RESOURCE_TYPE FlexPRET
  (* Standard: 61499-2 *)
  (* Version 0.1, 2016-00-28, hpea485, UOA *)
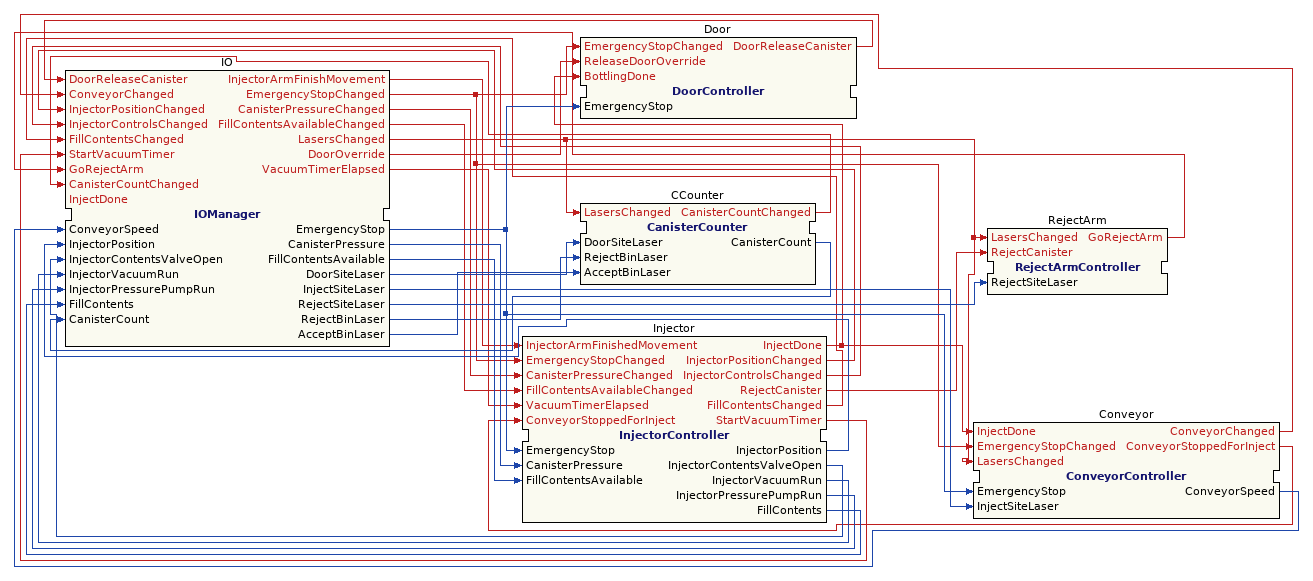
  FBS
    IO : IOManager;
    CCounter : CanisterCounter;
    Door : DoorController;
    Injector : InjectorController;
    Conveyor : ConveyorController;
    RejectArm : RejectArmController;
  END_FBS
  EVENT_CONNECTIONS
    IO.InjectorArmFinishMovement TO Injector.InjectorArmFinishedMovement;
    IO.EmergencyStopChanged TO Door.EmergencyStopChanged;
    IO.EmergencyStopChanged TO Injector.EmergencyStopChanged;
    IO.EmergencyStopChanged TO Conveyor.EmergencyStopChanged;
    IO.CanisterPressureChanged TO Injector.CanisterPressureChanged;
    IO.FillContentsAvailableChanged TO Injector.FillContentsAvailableChanged;
    IO.LasersChanged TO CCounter.LasersChanged;
    IO.LasersChanged TO RejectArm.LasersChanged;
    IO.LasersChanged TO Conveyor.LasersChanged;
    IO.DoorOverride TO Door.ReleaseDoorOverride;
    IO.VacuumTimerElapsed TO Injector.VacuumTimerElapsed;
    CCounter.CanisterCountChanged TO IO.CanisterCountChanged;
    Door.DoorReleaseCanister TO IO.DoorReleaseCanister;
    Injector.InjectDone TO Door.BottlingDone;
    Injector.InjectDone TO Conveyor.InjectDone;
    Injector.InjectorPositionChanged TO IO.InjectorPositionChanged;
    Injector.InjectorControlsChanged TO IO.InjectorControlsChanged;
    Injector.RejectCanister TO RejectArm.RejectCanister;
    Injector.FillContentsChanged TO IO.FillContentsChanged;
    Injector.StartVacuumTimer TO IO.StartVacuumTimer;
    Conveyor.ConveyorChanged TO IO.ConveyorChanged;
    Conveyor.ConveyorStoppedForInject TO Injector.ConveyorStoppedForInject;
    RejectArm.GoRejectArm TO IO.GoRejectArm;
  END_CONNECTIONS
  DATA_CONNECTIONS
    IO.EmergencyStop TO Door.EmergencyStop;
    IO.EmergencyStop TO Injector.EmergencyStop;
    IO.EmergencyStop TO Conveyor.EmergencyStop;
    IO.CanisterPressure TO Injector.CanisterPressure;
    IO.FillContentsAvailable TO Injector.FillContentsAvailable;
    IO.DoorSiteLaser TO CCounter.DoorSiteLaser;
    IO.InjectSiteLaser TO Conveyor.InjectSiteLaser;
    IO.RejectSiteLaser TO RejectArm.RejectSiteLaser;
    IO.RejectBinLaser TO CCounter.RejectBinLaser;
    IO.AcceptBinLaser TO CCounter.AcceptBinLaser;
    CCounter.CanisterCount TO IO.CanisterCount;
    Injector.InjectorPosition TO IO.InjectorPosition;
    Injector.InjectorContentsValveOpen TO IO.InjectorContentsValveOpen;
    Injector.InjectorVacuumRun TO IO.InjectorVacuumRun;
    Injector.InjectorPressurePumpRun TO IO.InjectorPressurePumpRun;
    Injector.FillContents TO IO.FillContents;
    Conveyor.ConveyorSpeed TO IO.ConveyorSpeed;
  END_CONNECTIONS
END_RESOURCE_TYPE
